RoboDK station: color_iden.rdk

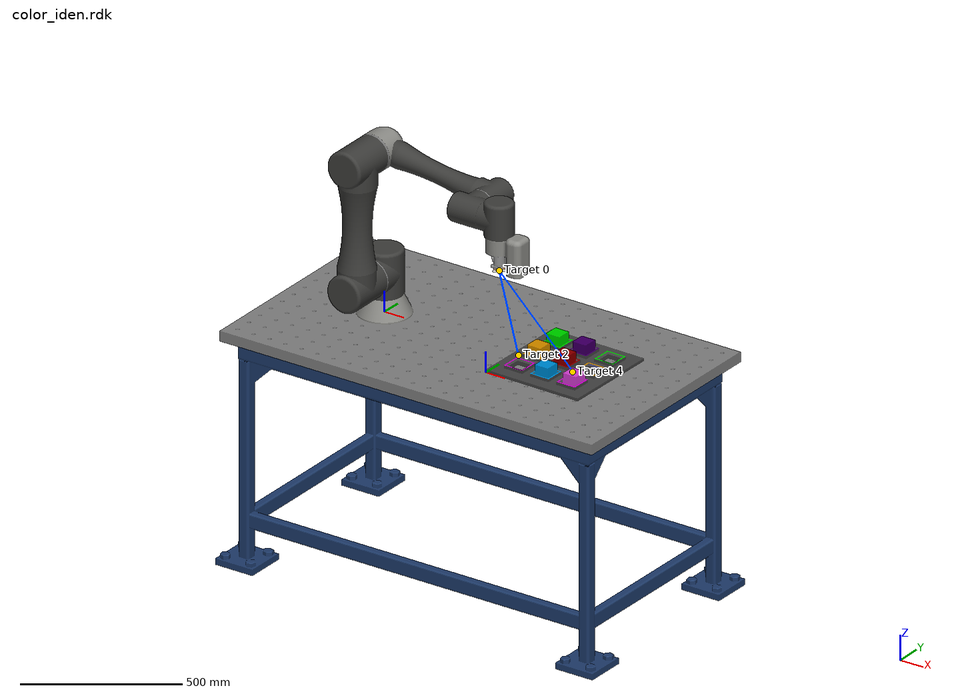
[picture v0: the station drawn from its stored meshes, robots at their saved joint values, targets as dots, program paths as lines]
Station New Station (1) (saved by RoboDK 5.9.2). Poses are relative to the parent item; angles as X-Y-Z fixed-axis rotations.
  - frame TM5-900 Base at (0, 0, 0) mm
    - robot TM5-900: 6 axes, payload 4 kg, reach 900 mm, repeatability 0.1 mm, weight 30 kg
        modified DH rows (alpha deg, a mm, theta deg, d mm): 0, 0, 0, 145.2; 90, 0, 90, 0; 0, 429, 0, 0; 0, 411, -90, 122.3; -90, 0, 0, 106.5; 90, 0, 180, 114.15
        joint limits [-360, -180, -155, -180, -180, -270] to [360, 180, 155, 180, 180, 270]; home [0, 0, 90, -90, 90, 0]; saved at [0, 0.638, 98.105, -8.743, 90, 0]
      - tool SMC ZXP7A01-ZP25C-X1 Vacuum Gripper, TCP at (0, 0, 62.5) mm, size 44 x 53.4 x 64 mm
  - object Table 1400x800x800mm at (0, 0, 0) mm, size 1420 x 820 x 800 mm, geometry from Table-1400x800x800mm.sld
  - frame Reference Frame at (500, -170, 0) mm, rotated rx 0 ry 0 rz -0.72 deg
    - object Pallete  at (0, 0, 0) mm, size 350 x 350 x 20 mm, geometry from Pallete .step
    - object Cube 50mm 2 at (50, 150, 0) mm, size 50 x 50 x 50 mm, geometry from Cube-50mm.sld
    - object Cube 50mm 3 at (50, 250, 0) mm, size 50 x 50 x 50 mm, geometry from Cube-50mm.sld
    - object Cube 50mm 4 at (150, 250, 0) mm, size 50 x 50 x 50 mm, geometry from Cube-50mm.sld
    - object Cube 50mm 5 at (150, 150, 0) mm, size 50 x 50 x 50 mm, geometry from Cube-50mm.sld
    - object Cube 50mm 6 at (150, 50, 0) mm, size 50 x 50 x 50 mm, geometry from Cube-50mm.sld
    - target Target 0 (Cartesian target) at (16.9, 47.92, 335.05) mm, rotated rx 180 ry 0 rz 90.72 deg; joints [0, 0, 90, 0, 90, 0] of TM5-900
    - target Target 2 (Cartesian target) at (71.58, 73.61, 50) mm, rotated rx 180 ry 0 rz 90.72 deg; joints [2.512, 25.678, 112.269, -47.948, 90, 2.512] of TM5-900
    - target Target 3 (Cartesian target) at (16.9, 47.92, 335.05) mm, rotated rx 180 ry 0 rz 90.72 deg; joints [0, 0.638, 98.105, -8.743, 90, 0] of TM5-900
    - target Target 4 (Cartesian target) at (276.56, 76.2, 50.05) mm, rotated rx 180 ry 0 rz 90.72 deg; joints [1.846, 47.126, 73.664, -30.79, 90, 1.846] of TM5-900
    - target Target 5 (Cartesian target) at (16.9, 47.92, 335.05) mm, rotated rx 180 ry 0 rz 90.72 deg; joints [0, 0.638, 98.105, -8.743, 90, 0] of TM5-900
  - program Prog1 (9 instructions, listed below)
  - program Prog2 (4 instructions, listed below)
  - object Cube 50mm at (755.63, -120.64, 0.05) mm, rotated rx 0 ry 0 rz -0.72 deg, size 50 x 50 x 50 mm, geometry from Cube-50mm.sld
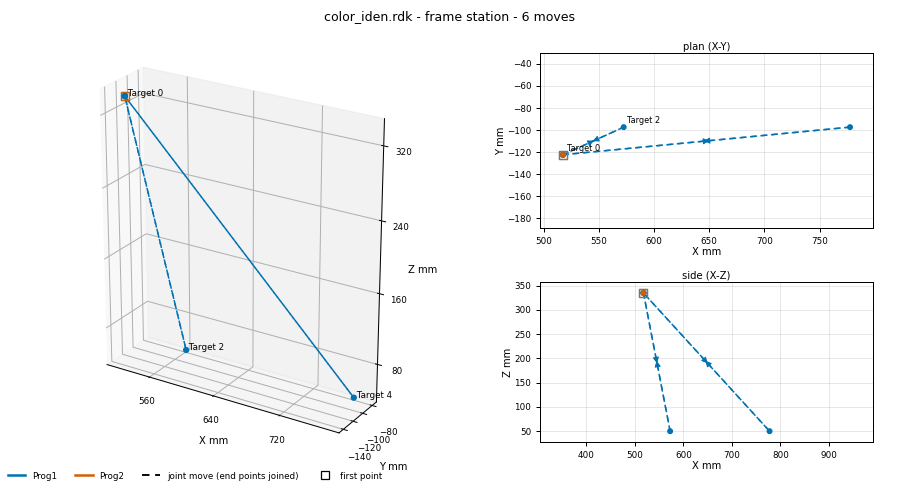
[picture p0: tool path of color_iden.rdk in frame station, 6 of 6 moves have a stored position in this frame; points joined in program order, loops and branches not executed]

--- program Prog1 (robot TM5-900) ---
  Set Ref.: Reference Frame
  Set Tool: SMC ZXP7A01-ZP25C-X1 Vacuum Gripper
  MoveJ (Target 0)
  MoveJ (Target 2)
  Attach to SMC ZXP7A01-ZP25C-X1 Vacuum Gripper
  MoveJ (Target 3)
  MoveJ (Target 4)
  Detach from SMC ZXP7A01-ZP25C-X1 Vacuum Gripper
  MoveJ (Target 5)

--- program Prog2 (robot TM5-900) ---
  Set Ref.: Reference Frame
  Set Tool: SMC ZXP7A01-ZP25C-X1 Vacuum Gripper
  MoveJ (Target 0)
  Replace objects
